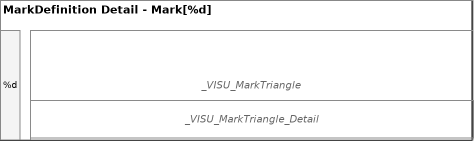
VISUALIZATION _VISU_MarkDefinition_Details  // 474x141
VAR_IN_OUT
	mInst : FB_MarkDefinition;
END_VAR
    Rectangle (0,0 472x141)
    Rectangle (0,0 234x20), "MarkDefinition Detail - Mark[%d]", text variable: mInst.nSelMark
    Frame (30,100 444x38)
        shows _VISU_MarkTriangle_Detail(mInst := mInst.pSelMark^)
    Frame (30,30 443x110)
        shows _VISU_MarkTriangle(mInst := mInst.pSelMark^)
    Scrollbar (0,30 20x110), "%d", text variable: mInst.nSelMark
        p2245068023: mInst._nMarks
        p1057716461: mInst.nSelMark
END_VISUALIZATION

(* stored: Version 1.1.0.1, ProductVersion 3.1.4024.11
   Visu _VISU_MarkDefinition_Details: Id {1825a0d1-06ed-46d6-808c-456191c63f56} *)
